// TIA Portal V20 export
TYPE "LKinCtrl_PathEditor_typePathTableUndoBuffer"
// stored: Access Published
   STRUCT
      stepsUndo { ExternalAccessible := 'False'; ExternalVisible := 'False'; ExternalWritable := 'False'} : Int;   // Total number of undos in both buffers
      stepsRedo { ExternalAccessible := 'False'; ExternalVisible := 'False'; ExternalWritable := 'False'} : Int;   // Total number of redos in both buffers
      pathBuffer { ExternalAccessible := 'False'; ExternalVisible := 'False'; ExternalWritable := 'False'} : Struct   // Path buffer, can reference command buffer.
         stepsUndo : Int;   // Number of possible undos in this buffer
         stepsRedo : Int;   // Number of possible redos in this buffers
         head : DInt;   // Pointer to first entry in path buffer
         entries : Array[1.."LKINCTRL_NO_OF_PATH_UNDOS_PATH_EDITOR"] of Struct   // Entries in path buffer
            pathNo : DInt;   // Selected path of entry
            commandNoUndo : DInt;   // Selected command when entry was saved
            commandNoRedo : DInt;   // Selected command after entry was saved
            commands : Array[1.."LKINCTRL_NO_OF_PATHDATA_ELEMENTS"] of "LKinCtrl_typePathDataElement";   // Commands of path
            nextType : USInt;   // Type of next entry. Path buffer, command buffer or end.
         END_STRUCT;
      END_STRUCT;
      commandBuffer { ExternalAccessible := 'False'; ExternalVisible := 'False'; ExternalWritable := 'False'} : Struct   // Command buffer, can be referenced by path buffer.
         stepsUndo : Int;   // Number of possible undos in this buffer
         stepsRedo : Int;   // Number of possible redos in this buffers
         head : DInt;   // Pointer to first entry in buffer buffer
         pathNo : DInt;   // Selected path of command
         commandNo : DInt;   // Selected command when entry was saved
         commands : Array[1.."LKINCTRL_NO_OF_COMMAND_UNDOS_PATH_EDITOR"] of "LKinCtrl_typePathDataElement";   // Entries in command buffer
      END_STRUCT;
   END_STRUCT;
END_TYPE
